SYSTEM BasicIcaruIo2 (* System Configuration *)
  (* Standard: 61499-1 *)
  (* Version 0.4, 2009-03-05, JHC, Holobloc Inc., Deleted Application. *)
  (* Version 0.3, 2003-12-05, JHC, Rockwell Automation, Renamed from NEWSYSTEM. *)
  (* Version 0.2, 2002-11-05, JHC, Rockwell Automation, Fixed missing (empty) FBD in Application. *)
  (* Version 0.1, 2002-01-17, JHC, Rockwell Automation, Minor cleanup *)
  (* Version 0.0, 2000-05-27, JHC, Rockwell Automation *)
  DEVICE ICARU4442 : RMT_DEV(MGR_ID := "localhost:61494")
    RESOURCE RESM : EMB_RES
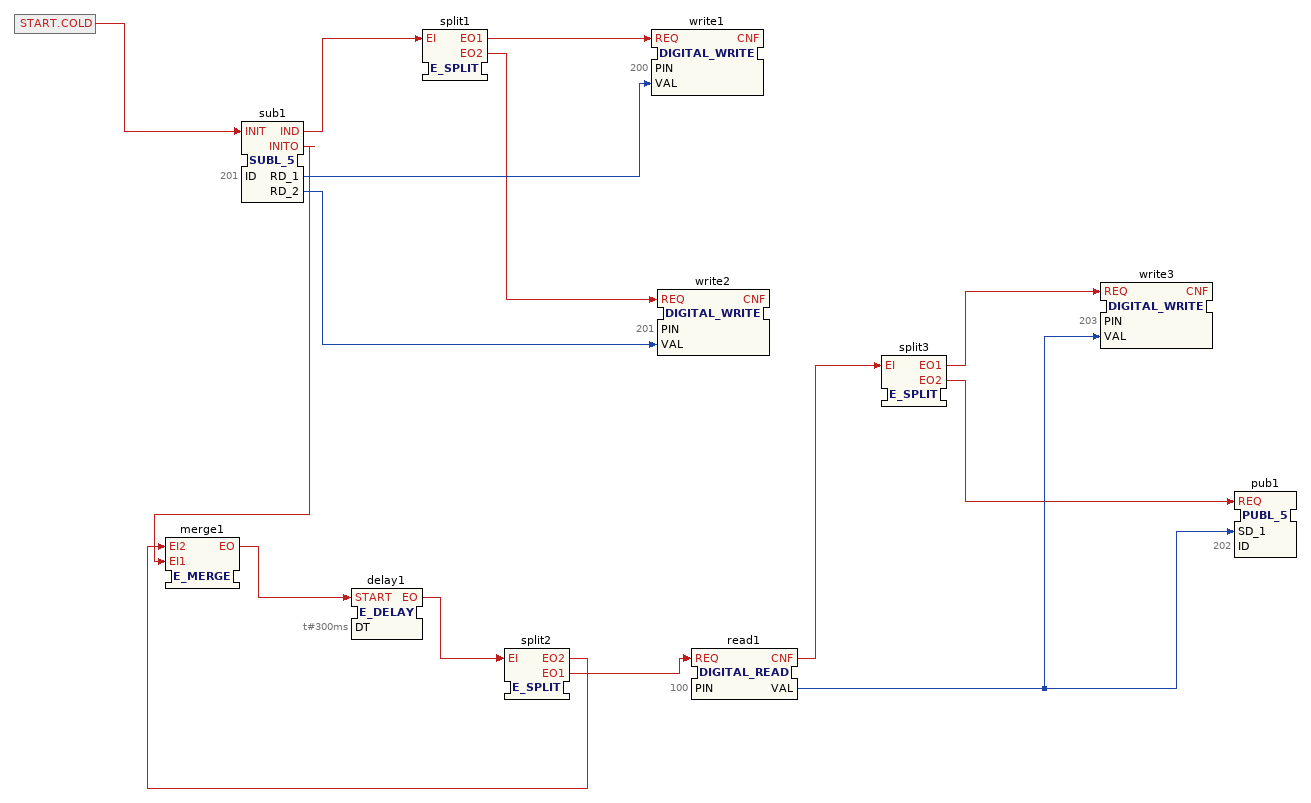
      FBS
        write1 : DIGITAL_WRITE(PIN := 200);
        split1 : E_SPLIT;
        write2 : DIGITAL_WRITE(PIN := 201);
        sub1 : SUBL_5(ID := 201);
        delay1 : E_DELAY(DT := t#300ms);
        merge1 : E_MERGE;
        split2 : E_SPLIT;
        read1 : DIGITAL_READ(PIN := 100);
        pub1 : PUBL_5(ID := 202);
        write3 : DIGITAL_WRITE(PIN := 203);
        split3 : E_SPLIT;
      END_FBS
      EVENT_CONNECTIONS
        split1.EO1 TO write1.REQ;
        split1.EO2 TO write2.REQ;
        START.COLD TO sub1.INIT;
        sub1.IND TO split1.EI;
        merge1.EO TO delay1.START;
        delay1.EO TO split2.EI;
        split2.EO2 TO merge1.EI2;
        split2.EO1 TO read1.REQ;
        read1.CNF TO split3.EI;
        split3.EO1 TO write3.REQ;
        split3.EO2 TO pub1.REQ;
        sub1.INITO TO merge1.EI1;
      END_CONNECTIONS
      DATA_CONNECTIONS
        sub1.RD_1 TO write1.VAL;
        sub1.RD_2 TO write2.VAL;
        read1.VAL TO pub1.SD_1;
        read1.VAL TO write3.VAL;
      END_CONNECTIONS
    END_RESOURCE
  END_DEVICE
  DEVICE DEV_CONTROL : FRAME_DEVICE(BOUNDS := [250,100,150,200], GRID := [1,5])
    RESOURCE RES1 : PANEL_RESOURCE(ROWS := 5)
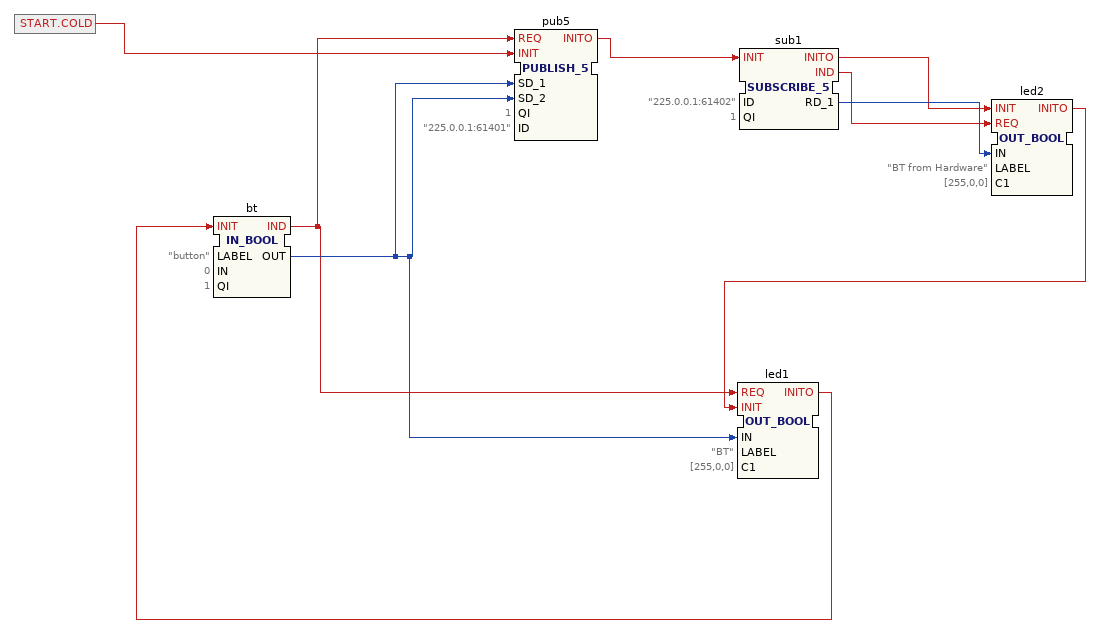
      FBS
        bt : IN_BOOL(LABEL := "button", IN := 0, QI := 1);
        led1 : OUT_BOOL(LABEL := "BT", C1 := [255,0,0]);
        pub5 : PUBLISH_5(QI := 1, ID := "225.0.0.1:61401");
        sub1 : SUBSCRIBE_5(ID := "225.0.0.1:61402", QI := 1);
        led2 : OUT_BOOL(LABEL := "BT from Hardware", C1 := [255,0,0]);
      END_FBS
      EVENT_CONNECTIONS
        bt.IND TO led1.REQ;
        bt.IND TO pub5.REQ;
        START.COLD TO pub5.INIT;
        led1.INITO TO bt.INIT;
        pub5.INITO TO sub1.INIT;
        sub1.INITO TO led2.INIT;
        led2.INITO TO led1.INIT;
        sub1.IND TO led2.REQ;
      END_CONNECTIONS
      DATA_CONNECTIONS
        bt.OUT TO led1.IN;
        bt.OUT TO pub5.SD_1;
        bt.OUT TO pub5.SD_2;
        sub1.RD_1 TO led2.IN;
      END_CONNECTIONS
    END_RESOURCE
  END_DEVICE
END_SYSTEM
